// TIA Portal V16 export
// export: Created 2021-04-11T09:51:31.8488981Z, ExportSetting WithDefaults, DisplayName Totally Integrated Automation Portal, DisplayVersion V16, DisplayName TIA Portal Version Control Interface, DisplayVersion V16, DisplayName TIA Portal Openness, DisplayVersion V16, DisplayName STEP 7 Professional, DisplayVersion V16, DisplayName STEP 7 Safety, DisplayVersion V16, DisplayName WinCC Unified SCADA Engineering System, DisplayVersion V16
VAR_GLOBAL   // PLC tag table "output"
   lampBlue AT %Q0.0 : Bool;   // Синяя лампа
   lampGreen AT %Q0.1 : Bool;   // Зеленая лампа
   lampRed AT %Q0.2 : Bool;   // Красная лампа
   qOn_ControlCurcuit AT %Q0.3 : Bool;   // включение цепей управления
   Y1q_ReadyDoze AT %Q0.4 : Bool;   // УП1 - доза готова
   Y2q_ReadyDoze AT %Q0.5 : Bool;   // УП2 - доза готова
   Conv1_FRV AT %Q0.6 : Bool;   // Конвейер1 - вперед
   Conv1_REV AT %Q0.7 : Bool;   // Конвейер1 - назад
   Conv2_FRV AT %Q1.0 : Bool;   // Конвейер2 - вперед
   Conv2_REV AT %Q1.1 : Bool;   // Конвейер2 - назад
   qDoor1_open AT %Q8.0 : Bool;   // Лопатка - открыть - 1
   qDoor1_close AT %Q8.1 : Bool;   // Лопатка - закрыть- 1
   qDoor2_open AT %Q8.2 : Bool;   // Лопатка - открыть - 2
   qDoor2_close AT %Q8.3 : Bool;   // Лопатка - закрыть- 2
   qDoor3_open AT %Q8.4 : Bool;   // Лопатка - открыть - 3
   qDoor3_close AT %Q8.5 : Bool;   // Лопатка - закрыть- 3
   qDoor4_open AT %Q8.6 : Bool;   // Лопатка - открыть - 4
   qDoor4_close AT %Q8.7 : Bool;   // Лопатка - закрыть- 4
   qDoor5_open AT %Q9.0 : Bool;   // Лопатка - открыть - 5
   qDoor5_close AT %Q9.1 : Bool;   // Лопатка - закрыть- 5
   qDoor6_open AT %Q9.2 : Bool;   // Лопатка - открыть - 6
   qDoor6_close AT %Q9.3 : Bool;   // Лопатка - закрыть- 6
   qDoor7_open AT %Q9.4 : Bool;   // Лопатка - открыть - 7
   qDoor7_close AT %Q9.5 : Bool;   // Лопатка - закрыть- 7
   qDoor8_open AT %Q9.6 : Bool;   // Лопатка - открыть - 8
   qDoor8_close AT %Q9.7 : Bool;   // Лопатка - закрыть- 8
   qBunker3_leftOpen AT %Q12.0 : Bool;   // Бункер - открыть влево - 3
   qBunker3_leftClose AT %Q12.1 : Bool;   // Бункер - закрыть влево - 3
   qBunker3_rightOpen AT %Q12.2 : Bool;   // Бункер - открыть вправо- 3
   qBunker3_rightClose AT %Q12.3 : Bool;   // Бункер - закрыть вправо- 3
   qBunker4_leftOpen AT %Q12.4 : Bool;   // Бункер - открыть влево - 4
   qBunker4_leftClose AT %Q12.5 : Bool;   // Бункер - закрыть влево - 4
   qBunker4_rightOpen AT %Q12.6 : Bool;   // Бункер - открыть вправо- 4
   qBunker4_rightClose AT %Q12.7 : Bool;   // Бункер - закрыть вправо- 4
   qBunker5_leftOpen AT %Q13.0 : Bool;   // Бункер - открыть влево - 5
   qBunker5_leftClose AT %Q13.1 : Bool;   // Бункер - закрыть влево - 5
   qBunker5_rightOpen AT %Q13.2 : Bool;   // Бункер - открыть вправо- 5
   qBunker5_rightClose AT %Q13.3 : Bool;   // Бункер - закрыть вправо- 5
   qBunker6_leftOpen AT %Q13.4 : Bool;   // Бункер - открыть влево - 6
   qBunker6_leftClose AT %Q13.5 : Bool;   // Бункер - закрыть влево - 6
   qBunker6_rightOpen AT %Q13.6 : Bool;   // Бункер - открыть вправо- 6
   qBunker6_rightClose AT %Q13.7 : Bool;   // Бункер - закрыть вправо- 6
   qBunker7_leftOpen AT %Q14.0 : Bool;   // Бункер - открыть влево - 7
   qBunker7_leftClose AT %Q14.1 : Bool;   // Бункер - закрыть влево - 7
   qBunker7_rightOpen AT %Q14.2 : Bool;   // Бункер - открыть вправо- 7
   qBunker7_rightClose AT %Q14.3 : Bool;   // Бункер - закрыть вправо- 7
   qBunker8_leftOpen AT %Q14.4 : Bool;   // Бункер - открыть влево - 8
   qBunker8_leftClose AT %Q14.5 : Bool;   // Бункер - закрыть влево - 8
   qBunker8_rightOpen AT %Q14.6 : Bool;   // Бункер - открыть вправо- 8
   qBunker8_rightClose AT %Q14.7 : Bool;   // Бункер - закрыть вправо- 8
   qBunker9_leftOpen AT %Q15.0 : Bool;   // Бункер - открыть влево - 9
   qBunker9_leftClose AT %Q15.1 : Bool;   // Бункер - закрыть влево - 9
   qBunker9_rightOpen AT %Q15.2 : Bool;   // Бункер - открыть вправо- 9
   qBunker9_rightClose AT %Q15.3 : Bool;   // Бункер - закрыть вправо- 9
   setVibration AT %QW64 : Int;   // задание уровня вибрации
   qDoor9_open AT %Q10.0 : Bool;   // Лопатка - открыть - 9
   qDoor9_close AT %Q10.1 : Bool;   // Лопатка - закрыть- 9
   qDoor10_open AT %Q10.2 : Bool;   // Лопатка - открыть - 10
   qDoor10_close AT %Q10.3 : Bool;   // Лопатка - закрыть- 10
   qDoor11_open AT %Q10.4 : Bool;   // Лопатка - открыть - 11
   qDoor11_close AT %Q10.5 : Bool;   // Лопатка - закрыть- 11
   qDoor12_open AT %Q10.6 : Bool;   // Лопатка - открыть - 12
   qDoor12_close AT %Q10.7 : Bool;   // Лопатка - закрыть- 12
   qBunker1_leftOpen AT %Q11.0 : Bool;   // Бункер - открыть влево - 1
   qBunker1_leftClose AT %Q11.1 : Bool;   // Бункер - закрыть влево - 1
   qBunker1_rightOpen AT %Q11.2 : Bool;   // Бункер - открыть вправо - 1
   qBunker1_rightClose AT %Q11.3 : Bool;   // Бункер - закрыть вправо - 1
   qBunker2_leftOpen AT %Q11.4 : Bool;   // Бункер - открыть влево - 2
   qBunker2_leftClose AT %Q11.5 : Bool;   // Бункер - закрыть влево - 2
   qBunker2_rightOpen AT %Q11.6 : Bool;   // Бункер - открыть вправо - 2
   qBunker2_rightClose AT %Q11.7 : Bool;   // Бункер - закрыть вправо - 2
   qBunker11_leftOpen AT %Q16.0 : Bool;   // Бункер - открыть влево - 11
   qBunker11_leftClose AT %Q16.1 : Bool;   // Бункер - закрыть влево - 11
   qBunker11_rightOpen AT %Q16.2 : Bool;   // Бункер - открыть вправо- 11
   qBunker11_rightClose AT %Q16.3 : Bool;   // Бункер - закрыть вправо- 11
   qBunker12_leftOpen AT %Q16.4 : Bool;   // Бункер - открыть влево - 12
   qBunker12_leftClose AT %Q16.5 : Bool;   // Бункер - закрыть влево - 12
   qBunker12_rightOpen AT %Q16.6 : Bool;   // Бункер - открыть вправо- 12
   qBunker12_rightClose AT %Q16.7 : Bool;   // Бункер - закрыть вправо- 12
   qBunker10_leftOpen AT %Q15.4 : Bool;   // Бункер - открыть влево - 10
   qBunker10_leftClose AT %Q15.5 : Bool;   // Бункер - закрыть влево - 10
   qBunker10_rightOpen AT %Q15.6 : Bool;   // Бункер - открыть вправо- 10
   qBunker10_rightClose AT %Q15.7 : Bool;   // Бункер - закрыть вправо- 10
   qFlipperUp AT %Q17.0 : Bool;   // плавник поднять
   qFlipperDown AT %Q17.1 : Bool;   // плавник опустить
   qVibroLot7_On AT %Q18.2 : Bool;   // управление вибролотком 7
   qVibroLot8_On AT %Q18.3 : Bool;   // управление вибролотком 8
   qVibroLot9_On AT %Q18.4 : Bool;   // управление вибролотком 9
   qVibroLot10_On AT %Q18.5 : Bool;   // управление вибролотком 10
   qVibroLot11_On AT %Q18.6 : Bool;   // управление вибролотком 11
   qVibroLot12_On AT %Q18.7 : Bool;   // управление вибролотком 12
   qVibroLot6_On AT %Q18.1 : Bool;   // управление вибролотком 6
   qVibroLot5_On AT %Q18.0 : Bool;   // управление вибролотком 5
   qVibroLot1_On AT %Q17.4 : Bool;   // управление вибролотком 1
   qVibroLot2_On AT %Q17.5 : Bool;   // управление вибролотком 2
   qVibroLot3_On AT %Q17.6 : Bool;   // управление вибролотком 3
   qVibroLot4_On AT %Q17.7 : Bool;   // управление вибролотком 4
   qVibroTable1 AT %Q17.2 : Bool;   // управление вибростолом 1
   qVibrotable2 AT %Q17.3 : Bool;   // управление вибростолом 2
   setSpeedConv AT %QW66 : Int;   // задание скорости конвейера
   startSourceConveyer AT %Q19.0 : Bool;   // запуск питателя
END_VAR
